(* PLC project Programme MGS_v0.3.10_Simulation.project, CODESYS CODESYS V3.5 SP19 Patch 1 *)
(* stored: creationDateTime 2026-07-04T07:58:13.0570557, modificationDateTime 2026-07-04T07:53:26.301727 *)

TYPE E_DiagState : (DISABLED := 0, READY := 1, INIT := 2, MONITORING := 3, ERROR := 4);
END_TYPE
